// TIA Portal V20 export
DATA_BLOCK "BK08"   // DB315
// stored: MemoryReserve 100
   VAR
      "X10-1.CATHODE MAIN P&P2 Z-AXIS LIMIT SENSOR(-)" : Bool := TRUE;
      "X10-2.CATHODE MAIN P&P2 Z-AXIS HOME SENSOR" : Bool := TRUE;
      "X12-1.CATHODE MAIN P&P2 Z-AXIS LIMIT SENSOR(+)" : Bool := TRUE;
      "X12-2.CATHODE MAIN P&P2 DETECT SENSOR" : Bool := FALSE;
      "X14-1.CATHODE MAIN P&P2 PRESSURE SWITCH" : Bool := FALSE;
      "X14-2.SPARE" : Bool := FALSE;
      "X16-1.SPARE" : Bool := FALSE;
      "X16-2.SPARE" : Bool := FALSE;
   END_VAR
BEGIN
END_DATA_BLOCK
